KUKA KRL program: Rack_Verde_Dejar.src, Rack_Verde_Dejar.dat

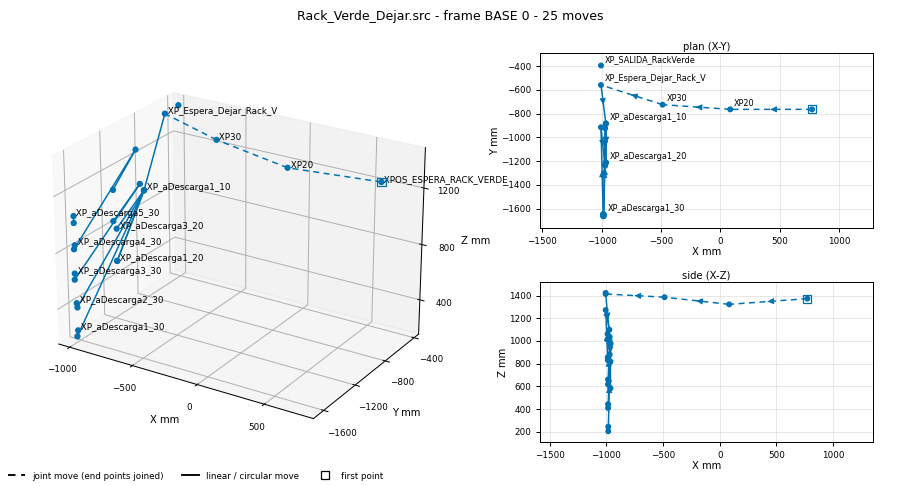
[picture p0: tool path of Rack_Verde_Dejar.src in frame BASE 0, 25 of 38 moves have a stored position in this frame; points joined in program order, loops and branches not executed]
--- Rack_Verde_Dejar.src ---
&ACCESS RVO1
&REL 3309
&COMMENT DEJAR BAT EN RACK VERDE
&PARAM EDITMASK = *
&PARAM TEMPLATE = C:\KRC\Roboter\Template\vorgabe
&PARAM DISKPATH = KRC:\R1\Program\MAFELEC
DEF Rack_Verde_Dejar( )
;FOLD INI;%{PE}
;FOLD BASISTECH INI
    GLOBAL INTERRUPT DECL 3 WHEN $STOPMESS==TRUE DO IR_STOPM ( )
    INTERRUPT ON 3
    BAS (#INITMOV,0 )
  ;ENDFOLD (BASISTECH INI)
;FOLD SPOTTECH INI
USERSPOT(#INIT)
;ENDFOLD (SPOTTECH INI)
;FOLD GRIPPERTECH INI
USER_GRP(0,DUMMY,DUMMY,GDEFAULT)
;ENDFOLD (GRIPPERTECH INI)
;FOLD USER INI
GIRO_A_P=FALSE
GIRO_A_N=FALSE
GIRO_B_P=FALSE
GIRO_B_N=FALSE
GIRO_C_P=FALSE
GIRO_C_N=FALSE
INTERRUPT DECL 26 WHEN I_121R1S102 OR I_121R1S202 DO PARO_RAPIDO ()
INTERRUPT DECL 27 WHEN I_121R1S302 OR I_121R1S402 DO PARO_RAPIDO ()
O_TYPE_INFO=0
SELECT_T1=FALSE

  ;ENDFOLD (USER INI)
;ENDFOLD (INI)
;################################################
; PROYECTO: MAFELEC PLANTA DE BATERIAS
; ROBOT: 121_R1
; PROGRAMA: DESCARGA DE BATERIA EN RACK VERDE
; CREADO POR: Tu amigo y vecino Spiderman(zaisor robotics)
; FECHA: 23-NOVIEMBRE-2022
; MODIFICADO POR:
; FECHA MODIFICACION: 17-ENERO-2023
;################################################

; FOLD CARGA VALORES DE POSICION

XP_DEJAR_VERDE=FRAME_POS
XP_DEJAR_VERDE.z=FRAME_POS.z+3
XP_DROP_1=XP_DEJAR_VERDE
XP_DROP_2=XP_DEJAR_VERDE
XP_DROP_3=XP_DEJAR_VERDE
XP_DROP_4=XP_DEJAR_VERDE
XP_DROP_5=XP_DEJAR_VERDE

XP_DROP_1.z=XP_DROP_1.z + 80
XP_DROP_2.z=XP_DROP_2.z + 80
XP_DROP_3.z=XP_DROP_3.z + 80
XP_DROP_4.z=XP_DROP_4.z + 80
XP_DROP_5.z=XP_DROP_5.z + 80
;ENDFOLD

;FOLD PTP POS_ESPERA_RACK_VERDE Vel=100 % H Tool[11]:T_Gripper1_Carga Base[0];%{PE}%R 8.3.48,%MKUKATPBASIS,%CMOVE,%VPTP,%P 1:PTP, 2:POS_ESPERA_RACK_VERDE, 3:, 5:100, 7:H
$BWDSTART=FALSE
PDAT_ACT=PH
FDAT_ACT=FPOS_ESPERA_RACK_VERDE
BAS(#PTP_PARAMS,100)
PTP XPOS_ESPERA_RACK_VERDE
;ENDFOLD
;ESPERA AREA 1
WAIT FOR I_ARDY_1
O_AREL_1=FALSE

Empujador(1,"R",TRUE)
Empujador(2,"R",TRUE)

;FOLD PTP P20 CONT Vel=100 % M Tool[11]:T_Gripper1_Carga Base[0];%{PE}%R 8.3.48,%MKUKATPBASIS,%CMOVE,%VPTP,%P 1:PTP, 2:P20, 3:C_DIS, 5:100, 7:M
$BWDSTART=FALSE
PDAT_ACT=PM
FDAT_ACT=FP20
BAS(#PTP_PARAMS,100)
PTP XP20 C_DIS
;ENDFOLD
;FOLD PTP P30 CONT Vel=100 % M Tool[11]:T_Gripper1_Carga Base[0];%{PE}%R 8.3.48,%MKUKATPBASIS,%CMOVE,%VPTP,%P 1:PTP, 2:P30, 3:C_DIS, 5:100, 7:M
$BWDSTART=FALSE
PDAT_ACT=PM
FDAT_ACT=FP30
BAS(#PTP_PARAMS,100)
PTP XP30 C_DIS
;ENDFOLD

; POSICION DE ESPERA A DEJAR BATERIA EN RACK VERDE
;FOLD PTP P_Espera_Dejar_Rack_V Vel=100 % L Tool[11]:T_Gripper1_Carga Base[0];%{PE}%R 8.3.48,%MKUKATPBASIS,%CMOVE,%VPTP,%P 1:PTP, 2:P_Espera_Dejar_Rack_V, 3:, 5:100, 7:L
$BWDSTART=FALSE
PDAT_ACT=PL
FDAT_ACT=FP_Espera_Dejar_Rack_V
BAS(#PTP_PARAMS,100)
PTP XP_Espera_Dejar_Rack_V
;ENDFOLD

; FOLD ACTIVA VIGILANCIA SOBREPASO
;INTERRUPT ON 26
;INTERRUPT ON 27
;ENDFOLD

;CONTROL DE AUSENCIA DE PIEZA EN GRIPPER
IF (I_SIMULACION==FALSE) THEN
IF NOT I_121R1S1000 THEN
HALT
ENDIF
ENDIF

;CONTROL APERTURA GRIPPER

IF (I_121R1S131A==FALSE) OR (I_121R1S132A==FALSE) OR (I_121R1S133A==FALSE) OR (I_121R1S134A==FALSE) THEN
HALT
ENDIF

IF PGNO==11 THEN
O_TYPE_RQ=TRUE
WAIT FOR (I_TYPE_INFO>10) AND (I_TYPE_INFO<16)
RV_Bandeja_Nr=I_TYPE_INFO
O_TYPE_RQ=FALSE
ENDIF

WAIT FOR (RV_Bandeja_Nr>10) AND (RV_Bandeja_Nr<16)

SWITCH RV_Bandeja_Nr ;

CASE 11
; MOVIMIENTOS HACIA BANDEJA 1
O_TYPE_INFO=11

WAIT FOR I_Rack1_S1==TRUE
;FOLD LIN P_aDescarga1_10 CONT Vel=0.5 m/s L Tool[11]:T_Gripper1_Carga Base[0];%{PE}%R 8.3.48,%MKUKATPBASIS,%CMOVE,%VLIN,%P 1:LIN, 2:P_aDescarga1_10, 3:C_DIS C_DIS, 5:0.5, 7:L
$BWDSTART=FALSE
LDAT_ACT=LL
FDAT_ACT=FP_aDescarga1_10
BAS(#CP_PARAMS,0.5)
LIN XP_aDescarga1_10 C_DIS C_DIS
;ENDFOLD
;FOLD LIN P_aDescarga1_20 CONT Vel=0.5 m/s L Tool[11]:T_Gripper1_Carga Base[0];%{PE}%R 8.3.48,%MKUKATPBASIS,%CMOVE,%VLIN,%P 1:LIN, 2:P_aDescarga1_20, 3:C_DIS C_DIS, 5:0.5, 7:L
$BWDSTART=FALSE
LDAT_ACT=LL
FDAT_ACT=FP_aDescarga1_20
BAS(#CP_PARAMS,0.5)
LIN XP_aDescarga1_20 C_DIS C_DIS
;ENDFOLD
O_LIMITS_OK=TRUE
O_LIMITS_NOK=FALSE

IF (O_INPICKER_OK==TRUE) AND (O_INPICKER_NOK==FALSE) AND (O_LIMITS_OK==TRUE) AND (O_LIMITS_NOK==FALSE) THEN
; #### MOVIMIENTOS A DESCARGA CONTROLADOS POR ####
; #### LA CAMARA DE VISION                    ####

;FOLD LIN P_DROP_1 Vel=0.3 m/s L Tool[11]:T_Gripper1_Carga Base[0];%{PE}%R 8.3.48,%MKUKATPBASIS,%CMOVE,%VLIN,%P 1:LIN, 2:P_DROP_1, 3:, 5:0.3, 7:L
$BWDSTART=FALSE
LDAT_ACT=LL
FDAT_ACT=FP_DROP_1
BAS(#CP_PARAMS,0.3)
LIN XP_DROP_1
;ENDFOLD
;FOLD LIN P_DEJAR_VERDE Vel=0.1 m/s L Tool[11]:T_Gripper1_Carga Base[0];%{PE}%R 8.3.48,%MKUKATPBASIS,%CMOVE,%VLIN,%P 1:LIN, 2:P_DEJAR_VERDE, 3:, 5:0.1, 7:L
$BWDSTART=FALSE
LDAT_ACT=LL
FDAT_ACT=FP_DEJAR_VERDE
BAS(#CP_PARAMS,0.1)
LIN XP_DEJAR_VERDE
;ENDFOLD

ELSE

; #### MOVIMIENTOS A DESCARGA CONTROLADOS POR ####
; #### EL OPERARIO                            ####
;FOLD ESPERA LLAVE SELECTORA EN MODO T1
WAIT FOR $T1
SELECT_T1=TRUE
;ENDFOLD
;FOLD LIN P_aDescarga1_30 CONT Vel=0.2 m/s L Tool[11]:T_Gripper1_Carga Base[0];%{PE}%R 8.3.48,%MKUKATPBASIS,%CMOVE,%VLIN,%P 1:LIN, 2:P_aDescarga1_30, 3:C_DIS C_DIS, 5:0.2, 7:L
$BWDSTART=FALSE
LDAT_ACT=LL
FDAT_ACT=FP_aDescarga1_30
BAS(#CP_PARAMS,0.2)
LIN XP_aDescarga1_30 C_DIS C_DIS
;ENDFOLD

;POSICION DE DESCARGA 1
;CUIDADO CON EL LINEAL NO EJECUTARLO HASTA EL FINAL
;POSIBILIDAD DE COLISION
;EN ESTE PUNTO LLEVAR EL ROBOT HASTA LA DESCARGA DE BANDEJA
;UNA VEZ TENEMOS EL ROBOT YA EN LA POSICION DE DEJADA TENEMOS
;QUE ACTIVAR LAS SALIDAS DE LAS CLAMPAS PARA DEJAR LA BATERIA
;SALIDA 246 O_121R1Y13A PINES BLOQUEO ADELANTE ESTARA EN 1 PONERLA A 0
;SEGUIDAMENTE LA SALIDA 245 O_121R1Y13B PINES BLOQUEO ATRAS ESTARA A 0 PONERLA A 1
;AL ABRIR LOS PINES DE LAS CLAMPAS EL SIGUIENTE PASO ES SELECCIONAR LA LINEA
;ENDIF Y CONTINUAR PROGRAMA
;FOLD LIN Rack_Verde_Pos1 Vel=0.2 m/s L Tool[11]:T_Gripper1_Carga Base[0];%{PE}%R 8.3.48,%MKUKATPBASIS,%CMOVE,%VLIN,%P 1:LIN, 2:Rack_Verde_Pos1, 3:, 5:0.2, 7:L
$BWDSTART=FALSE
LDAT_ACT=LL
FDAT_ACT=FRack_Verde_Pos1
BAS(#CP_PARAMS,0.2)
LIN XRack_Verde_Pos1
;ENDFOLD
ENDIF

CASE 12
; MOVIMIENTOS HACIA BANDEJA 2
O_TYPE_INFO=12
WAIT FOR I_Rack1_S2==TRUE
;FOLD LIN P_aDescarga2_10 CONT Vel=0.5 m/s L Tool[11]:T_Gripper1_Carga Base[0];%{PE}%R 8.3.48,%MKUKATPBASIS,%CMOVE,%VLIN,%P 1:LIN, 2:P_aDescarga2_10, 3:C_DIS C_DIS, 5:0.5, 7:L
$BWDSTART=FALSE
LDAT_ACT=LL
FDAT_ACT=FP_aDescarga2_10
BAS(#CP_PARAMS,0.5)
LIN XP_aDescarga2_10 C_DIS C_DIS
;ENDFOLD
;FOLD LIN P_aDescarga2_20 CONT Vel=0.5 m/s L Tool[11]:T_Gripper1_Carga Base[0];%{PE}%R 8.3.48,%MKUKATPBASIS,%CMOVE,%VLIN,%P 1:LIN, 2:P_aDescarga2_20, 3:C_DIS C_DIS, 5:0.5, 7:L
$BWDSTART=FALSE
LDAT_ACT=LL
FDAT_ACT=FP_aDescarga2_20
BAS(#CP_PARAMS,0.5)
LIN XP_aDescarga2_20 C_DIS C_DIS
;ENDFOLD

IF (O_INPICKER_OK==TRUE) AND (O_INPICKER_NOK==FALSE) AND (O_LIMITS_OK==TRUE) AND (O_LIMITS_NOK==FALSE) THEN
; #### MOVIMIENTOS A DESCARGA CONTROLADOS POR ####
; #### LA CAMARA DE VISION                    ####

;FOLD LIN P_DROP_2 Vel=0.3 m/s L Tool[11]:T_Gripper1_Carga Base[0];%{PE}%R 8.3.48,%MKUKATPBASIS,%CMOVE,%VLIN,%P 1:LIN, 2:P_DROP_2, 3:, 5:0.3, 7:L
$BWDSTART=FALSE
LDAT_ACT=LL
FDAT_ACT=FP_DROP_2
BAS(#CP_PARAMS,0.3)
LIN XP_DROP_2
;ENDFOLD
;FOLD LIN P_DEJAR_VERDE Vel=0.1 m/s L Tool[11]:T_Gripper1_Carga Base[0];%{PE}%R 8.3.48,%MKUKATPBASIS,%CMOVE,%VLIN,%P 1:LIN, 2:P_DEJAR_VERDE, 3:, 5:0.1, 7:L
$BWDSTART=FALSE
LDAT_ACT=LL
FDAT_ACT=FP_DEJAR_VERDE
BAS(#CP_PARAMS,0.1)
LIN XP_DEJAR_VERDE
;ENDFOLD

ELSE
; #### MOVIMIENTOS A DESCARGA CONTROLADOS POR ####
; #### EL OPERARIO                            ####
;FOLD ESPERA LLAVE SELECTORA EN MODO T1
WAIT FOR $T1
SELECT_T1=TRUE
;ENDFOLD
;FOLD LIN P_aDescarga2_30 CONT Vel=0.2 m/s L Tool[11]:T_Gripper1_Carga Base[0];%{PE}%R 8.3.48,%MKUKATPBASIS,%CMOVE,%VLIN,%P 1:LIN, 2:P_aDescarga2_30, 3:C_DIS C_DIS, 5:0.2, 7:L
$BWDSTART=FALSE
LDAT_ACT=LL
FDAT_ACT=FP_aDescarga2_30
BAS(#CP_PARAMS,0.2)
LIN XP_aDescarga2_30 C_DIS C_DIS
;ENDFOLD

;POSICION DE DESCARGA 2
;CUIDADO CON EL LINEAL NO EJECUTARLO HASTA EL FINAL
;POSIBILIDAD DE COLISION
;EN ESTE PUNTO LLEVAR EL ROBOT HASTA LA DESCARGA DE BANDEJA
;UNA VEZ TENEMOS EL ROBOT YA EN LA POSICION DE DEJADA TENEMOS
;QUE ACTIVAR LAS SALIDAS DE LAS CLAMPAS PARA DEJAR LA BATERIA
;SALIDA 246 O_121R1Y13A PINES BLOQUEO ADELANTE ESTARA EN 1 PONERLA A 0
;SEGUIDAMENTE LA SALIDA 245 O_121R1Y13B PINES BLOQUEO ATRAS ESTARA A 0 PONERLA A 1
;AL ABRIR LOS PINES DE LAS CLAMPAS EL SIGUIENTE PASO ES SELECCIONAR LA LINEA
;ENDIF Y CONTINUAR PROGRAMA
;FOLD LIN Rack_Verde_Pos2 Vel=0.2 m/s L Tool[11]:T_Gripper1_Carga Base[0];%{PE}%R 8.3.48,%MKUKATPBASIS,%CMOVE,%VLIN,%P 1:LIN, 2:Rack_Verde_Pos2, 3:, 5:0.2, 7:L
$BWDSTART=FALSE
LDAT_ACT=LL
FDAT_ACT=FRack_Verde_Pos2
BAS(#CP_PARAMS,0.2)
LIN XRack_Verde_Pos2
;ENDFOLD
ENDIF

CASE 13
; MOVIMIENTOS HACIA BANDEJA 3
O_TYPE_INFO=13
WAIT FOR I_Rack1_S3==TRUE
;FOLD LIN P_aDescarga3_10 CONT Vel=0.5 m/s L Tool[11]:T_Gripper1_Carga Base[0];%{PE}%R 8.3.48,%MKUKATPBASIS,%CMOVE,%VLIN,%P 1:LIN, 2:P_aDescarga3_10, 3:C_DIS C_DIS, 5:0.5, 7:L
$BWDSTART=FALSE
LDAT_ACT=LL
FDAT_ACT=FP_aDescarga3_10
BAS(#CP_PARAMS,0.5)
LIN XP_aDescarga3_10 C_DIS C_DIS
;ENDFOLD
;FOLD LIN P_aDescarga3_20 CONT Vel=0.5 m/s L Tool[11]:T_Gripper1_Carga Base[0];%{PE}%R 8.3.48,%MKUKATPBASIS,%CMOVE,%VLIN,%P 1:LIN, 2:P_aDescarga3_20, 3:C_DIS C_DIS, 5:0.5, 7:L
$BWDSTART=FALSE
LDAT_ACT=LL
FDAT_ACT=FP_aDescarga3_20
BAS(#CP_PARAMS,0.5)
LIN XP_aDescarga3_20 C_DIS C_DIS
;ENDFOLD


IF (O_INPICKER_OK==TRUE) AND (O_INPICKER_NOK==FALSE) AND (O_LIMITS_OK==TRUE) AND (O_LIMITS_NOK==FALSE) THEN
; #### MOVIMIENTOS A DESCARGA CONTROLADOS POR ####
; #### LA CAMARA DE VISION                    ####

;FOLD LIN P_DROP_3 Vel=0.3 m/s L Tool[11]:T_Gripper1_Carga Base[0];%{PE}%R 8.3.48,%MKUKATPBASIS,%CMOVE,%VLIN,%P 1:LIN, 2:P_DROP_3, 3:, 5:0.3, 7:L
$BWDSTART=FALSE
LDAT_ACT=LL
FDAT_ACT=FP_DROP_3
BAS(#CP_PARAMS,0.3)
LIN XP_DROP_3
;ENDFOLD
;FOLD LIN P_DEJAR_VERDE Vel=0.1 m/s L Tool[11]:T_Gripper1_Carga Base[0];%{PE}%R 8.3.48,%MKUKATPBASIS,%CMOVE,%VLIN,%P 1:LIN, 2:P_DEJAR_VERDE, 3:, 5:0.1, 7:L
$BWDSTART=FALSE
LDAT_ACT=LL
FDAT_ACT=FP_DEJAR_VERDE
BAS(#CP_PARAMS,0.1)
LIN XP_DEJAR_VERDE
;ENDFOLD

ELSE
; #### MOVIMIENTOS A DESCARGA CONTROLADOS POR ####
; #### EL OPERARIO                            ####
;FOLD ESPERA LLAVE SELECTORA EN MODO T1
WAIT FOR $T1
SELECT_T1=TRUE
;ENDFOLD
;FOLD LIN P_aDescarga3_30 CONT Vel=0.2 m/s L Tool[11]:T_Gripper1_Carga Base[0];%{PE}%R 8.3.48,%MKUKATPBASIS,%CMOVE,%VLIN,%P 1:LIN, 2:P_aDescarga3_30, 3:C_DIS C_DIS, 5:0.2, 7:L
$BWDSTART=FALSE
LDAT_ACT=LL
FDAT_ACT=FP_aDescarga3_30
BAS(#CP_PARAMS,0.2)
LIN XP_aDescarga3_30 C_DIS C_DIS
;ENDFOLD

;POSICION DE DESCARGA 3
;CUIDADO CON EL LINEAL NO EJECUTARLO HASTA EL FINAL
;POSIBILIDAD DE COLISION
;EN ESTE PUNTO LLEVAR EL ROBOT HASTA LA DESCARGA DE BANDEJA
;UNA VEZ TENEMOS EL ROBOT YA EN LA POSICION DE DEJADA TENEMOS
;QUE ACTIVAR LAS SALIDAS DE LAS CLAMPAS PARA DEJAR LA BATER
;SALIDA 246 y 248 PINES BLOQUEO ADELANTE ESTARA EN 1 PONERLA A 0
;SEGUIDAMENTE LA SALIDA 245 y 247 PINES BLOQUEO ATRAS ESTARA A 0 PONERLA A 1
;AL ABRIR LOS PINES DE LAS CLAMPAS EL SIGUIENTE PASO ES SELECCIONAR LA LINEA
;ENDIF Y CONTINUAR PROGRAMA
;FOLD LIN Rack_Verde_Pos3 Vel=0.2 m/s L Tool[11]:T_Gripper1_Carga Base[0];%{PE}%R 8.3.48,%MKUKATPBASIS,%CMOVE,%VLIN,%P 1:LIN, 2:Rack_Verde_Pos3, 3:, 5:0.2, 7:L
$BWDSTART=FALSE
LDAT_ACT=LL
FDAT_ACT=FRack_Verde_Pos3
BAS(#CP_PARAMS,0.2)
LIN XRack_Verde_Pos3
;ENDFOLD
ENDIF

CASE 14
; MOVIMIENTOS HACIA BANDEJA4
O_TYPE_INFO=14
WAIT FOR I_Rack1_S4==TRUE
;FOLD LIN P_aDescarga4_10 CONT Vel=0.5 m/s L Tool[11]:T_Gripper1_Carga Base[0];%{PE}%R 8.3.48,%MKUKATPBASIS,%CMOVE,%VLIN,%P 1:LIN, 2:P_aDescarga4_10, 3:C_DIS C_DIS, 5:0.5, 7:L
$BWDSTART=FALSE
LDAT_ACT=LL
FDAT_ACT=FP_aDescarga4_10
BAS(#CP_PARAMS,0.5)
LIN XP_aDescarga4_10 C_DIS C_DIS
;ENDFOLD
;FOLD LIN P_aDescarga4_20 CONT Vel=0.5 m/s L Tool[11]:T_Gripper1_Carga Base[0];%{PE}%R 8.3.48,%MKUKATPBASIS,%CMOVE,%VLIN,%P 1:LIN, 2:P_aDescarga4_20, 3:C_DIS C_DIS, 5:0.5, 7:L
$BWDSTART=FALSE
LDAT_ACT=LL
FDAT_ACT=FP_aDescarga4_20
BAS(#CP_PARAMS,0.5)
LIN XP_aDescarga4_20 C_DIS C_DIS
;ENDFOLD

IF (O_INPICKER_OK==TRUE) AND (O_INPICKER_NOK==FALSE) AND (O_LIMITS_OK==TRUE) AND (O_LIMITS_NOK==FALSE) THEN
; #### MOVIMIENTOS A DESCARGA CONTROLADOS POR ####
; #### LA CAMARA DE VISION                    ####

;FOLD LIN P_DROP_4 Vel=0.3 m/s L Tool[11]:T_Gripper1_Carga Base[0];%{PE}%R 8.3.48,%MKUKATPBASIS,%CMOVE,%VLIN,%P 1:LIN, 2:P_DROP_4, 3:, 5:0.3, 7:L
$BWDSTART=FALSE
LDAT_ACT=LL
FDAT_ACT=FP_DROP_4
BAS(#CP_PARAMS,0.3)
LIN XP_DROP_4
;ENDFOLD
;FOLD LIN P_DEJAR_VERDE Vel=0.1 m/s L Tool[11]:T_Gripper1_Carga Base[0];%{PE}%R 8.3.48,%MKUKATPBASIS,%CMOVE,%VLIN,%P 1:LIN, 2:P_DEJAR_VERDE, 3:, 5:0.1, 7:L
$BWDSTART=FALSE
LDAT_ACT=LL
FDAT_ACT=FP_DEJAR_VERDE
BAS(#CP_PARAMS,0.1)
LIN XP_DEJAR_VERDE
;ENDFOLD

ELSE
; #### MOVIMIENTOS A DESCARGA CONTROLADOS POR ####
; #### EL OPERARIO                            ####
;FOLD ESPERA LLAVE SELECTORA EN MODO T1
WAIT FOR $T1
SELECT_T1=TRUE
;ENDFOLD
;FOLD LIN P_aDescarga4_30 CONT Vel=0.2 m/s L Tool[11]:T_Gripper1_Carga Base[0];%{PE}%R 8.3.48,%MKUKATPBASIS,%CMOVE,%VLIN,%P 1:LIN, 2:P_aDescarga4_30, 3:C_DIS C_DIS, 5:0.2, 7:L
$BWDSTART=FALSE
LDAT_ACT=LL
FDAT_ACT=FP_aDescarga4_30
BAS(#CP_PARAMS,0.2)
LIN XP_aDescarga4_30 C_DIS C_DIS
;ENDFOLD

;POSICION DE DESCARGA 4
;CUIDADO CON EL LINEAL NO EJECUTARLO HASTA EL FINAL
;POSIBILIDAD DE COLISION
;EN ESTE PUNTO LLEVAR EL ROBOT HASTA LA DESCARGA DE BANDEJA
;UNA VEZ TENEMOS EL ROBOT YA EN LA POSICION DE DEJADA TENEMOS
;QUE ACTIVAR LAS SALIDAS DE LAS CLAMPAS PARA DEJAR LA BATERIA
;SALIDA 246 y 248 PINES BLOQUEO ADELANTE ESTARA EN 1 PONERLA A 0
;SEGUIDAMENTE LA SALIDA 245 y 247 PINES BLOQUEO ATRAS ESTARA A 0 PONERLA A 1
;AL ABRIR LOS PINES DE LAS CLAMPAS EL SIGUIENTE PASO ES SELECCIONAR LA LINEA
;ENDIF Y CONTINUAR PROGRAMA
;FOLD LIN Rack_Verde_Pos4 Vel=0.2 m/s L Tool[11]:T_Gripper1_Carga Base[0];%{PE}%R 8.3.48,%MKUKATPBASIS,%CMOVE,%VLIN,%P 1:LIN, 2:Rack_Verde_Pos4, 3:, 5:0.2, 7:L
$BWDSTART=FALSE
LDAT_ACT=LL
FDAT_ACT=FRack_Verde_Pos4
BAS(#CP_PARAMS,0.2)
LIN XRack_Verde_Pos4
;ENDFOLD
ENDIF

CASE 15
; MOVIMIENTOS HACIA BANDEJA 5
O_TYPE_INFO=15
WAIT FOR I_Rack1_S5==TRUE
;FOLD LIN P_aDescarga5_10 CONT Vel=0.5 m/s L Tool[11]:T_Gripper1_Carga Base[0];%{PE}%R 8.3.48,%MKUKATPBASIS,%CMOVE,%VLIN,%P 1:LIN, 2:P_aDescarga5_10, 3:C_DIS C_DIS, 5:0.5, 7:L
$BWDSTART=FALSE
LDAT_ACT=LL
FDAT_ACT=FP_aDescarga5_10
BAS(#CP_PARAMS,0.5)
LIN XP_aDescarga5_10 C_DIS C_DIS
;ENDFOLD
;FOLD LIN P_aDescarga5_20 CONT Vel=0.5 m/s L Tool[11]:T_Gripper1_Carga Base[0];%{PE}%R 8.3.48,%MKUKATPBASIS,%CMOVE,%VLIN,%P 1:LIN, 2:P_aDescarga5_20, 3:C_DIS C_DIS, 5:0.5, 7:L
$BWDSTART=FALSE
LDAT_ACT=LL
FDAT_ACT=FP_aDescarga5_20
BAS(#CP_PARAMS,0.5)
LIN XP_aDescarga5_20 C_DIS C_DIS
;ENDFOLD

IF (O_INPICKER_OK==TRUE) AND (O_INPICKER_NOK==FALSE) AND (O_LIMITS_OK==TRUE) AND (O_LIMITS_NOK==FALSE) THEN
; #### MOVIMIENTOS A DESCARGA CONTROLADOS POR ####
; #### LA CAMARA DE VISION                    ####

;FOLD LIN P_DROP_5 Vel=0.3 m/s L Tool[11]:T_Gripper1_Carga Base[0];%{PE}%R 8.3.48,%MKUKATPBASIS,%CMOVE,%VLIN,%P 1:LIN, 2:P_DROP_5, 3:, 5:0.3, 7:L
$BWDSTART=FALSE
LDAT_ACT=LL
FDAT_ACT=FP_DROP_5
BAS(#CP_PARAMS,0.3)
LIN XP_DROP_5
;ENDFOLD
;FOLD LIN P_DEJAR_VERDE Vel=0.1 m/s L Tool[11]:T_Gripper1_Carga Base[0];%{PE}%R 8.3.48,%MKUKATPBASIS,%CMOVE,%VLIN,%P 1:LIN, 2:P_DEJAR_VERDE, 3:, 5:0.1, 7:L
$BWDSTART=FALSE
LDAT_ACT=LL
FDAT_ACT=FP_DEJAR_VERDE
BAS(#CP_PARAMS,0.1)
LIN XP_DEJAR_VERDE
;ENDFOLD

ELSE
; #### MOVIMIENTOS A DESCARGA CONTROLADOS POR ####
; #### EL OPERARIO                            ####
;FOLD ESPERA LLAVE SELECTORA EN MODO T1
WAIT FOR $T1
SELECT_T1=TRUE
;ENDFOLD
;FOLD LIN P_aDescarga5_30 CONT Vel=0.2 m/s L Tool[11]:T_Gripper1_Carga Base[0];%{PE}%R 8.3.48,%MKUKATPBASIS,%CMOVE,%VLIN,%P 1:LIN, 2:P_aDescarga5_30, 3:C_DIS C_DIS, 5:0.2, 7:L
$BWDSTART=FALSE
LDAT_ACT=LL
FDAT_ACT=FP_aDescarga5_30
BAS(#CP_PARAMS,0.2)
LIN XP_aDescarga5_30 C_DIS C_DIS
;ENDFOLD

;POSICION DE DESCARGA 5
;CUIDADO CON EL LINEAL NO EJECUTARLO HASTA EL FINAL
;POSIBILIDAD DE COLISION
;EN ESTE PUNTO LLEVAR EL ROBOT HASTA LA DESCARGA DE BANDEJA
;UNA VEZ TENEMOS EL ROBOT YA EN LA POSICION DE DEJADA TENEMOS
;QUE ACTIVAR LAS SALIDAS DE LAS CLAMPAS PARA DEJAR LA BATERIA
;SALIDA 246 O_121R1Y13A PINES BLOQUEO ADELANTE ESTARA EN 1 PONERLA A 0
;SEGUIDAMENTE LA SALIDA 245 O_121R1Y13B PINES BLOQUEO ATRAS ESTARA A 0 PONERLA A 1
;AL ABRIR LOS PINES DE LAS CLAMPAS EL SIGUIENTE PASO ES SELECCIONAR LA LINEA
;ENDIF Y CONTINUAR PROGRAMA
;FOLD LIN Rack_Verde_Pos5 Vel=0.2 m/s L Tool[11]:T_Gripper1_Carga Base[0];%{PE}%R 8.3.48,%MKUKATPBASIS,%CMOVE,%VLIN,%P 1:LIN, 2:Rack_Verde_Pos5, 3:, 5:0.2, 7:L
$BWDSTART=FALSE
LDAT_ACT=LL
FDAT_ACT=FRack_Verde_Pos5
BAS(#CP_PARAMS,0.2)
LIN XRack_Verde_Pos5
;ENDFOLD
ENDIF

DEFAULT
HALT
HALT
; #### CODIGO DE DESCARGA ERRONEO ####
HALT
BRAKE
ENDSWITCH

; FOLD MOVIMIENTOS DE SALIDA RACK VERDE
INI_DROP:
GIRO_A_P=FALSE
GIRO_A_N=FALSE
GIRO_B_P=FALSE
GIRO_B_N=FALSE
GIRO_C_P=FALSE
GIRO_C_N=FALSE

PTP $POS_ACT

IF (I_SIMULACION==FALSE) THEN

Repite=0

WHILE (I_121R1S102==TRUE) OR (I_121R1S202==TRUE) OR (I_121R1S302==TRUE) OR (I_121R1S402==TRUE)

Repite=Repite+1
LIN_REL{Z +1}
WAIT SEC 0.1

IF Repite>=3 THEN
HALT
; SUPERADO NUMERO DE REPETICIONES
HALT
ENDIF

ENDWHILE

Repite=0

WHILE (I_121R1S101==FALSE) AND (I_121R1S201==FALSE) AND (I_121R1S301==FALSE) AND (I_121R1S401==FALSE)
IF (I_121R1S102==TRUE) OR (I_121R1S202==TRUE) OR (I_121R1S302==TRUE) OR (I_121R1S402==TRUE) THEN
HALT
HALT
HALT
ENDIF
Repite=Repite+1
LIN_REL{Z -1}
WAIT SEC 0.1

IF Repite>=8 THEN
HALT
; SUPERADO NUMERO DE REPETICIONES
HALT
ENDIF

;PARA ABRIR PINES DE LA BATERIA SALIDA O_121R1Y13B
;GOTO ctrl_dejar
ENDWHILE

; #### CONTROL DE PRESENCIA PARA ABRIR ####
WAIT FOR (I_121R1S101==TRUE) OR (I_121R1S301==TRUE) OR (I_121R1S201==TRUE) OR (I_121R1S401==TRUE)
fin_dejar:
ENDIF

O_INPICKER_OK=FALSE
O_INPICKER_NOK=FALSE
O_LIMITS_OK=FALSE
O_LIMITS_NOK=FALSE
O_LIMIT_X=FALSE
O_LIMIT_Y=FALSE
O_LIMIT_Z=FALSE
O_LIMIT_A=FALSE
O_LIMIT_B=FALSE
O_LIMIT_C=FALSE

PTP $POS_ACT
PINES("R")

PTP $POS_ACT
WAIT FOR $EXT; CAMBIAR LA LLAVE A MODO EXT

LIN_REL{Z +100}
O_JRDY_2=TRUE
BAS(#CP_PARAMS,1.5)

; #### CONTROL DE AUSENCIA DE BATERIA ####
WAIT FOR NOT I_121R1S1000

LIN_REL{Y 300,Z +100} C_DIS
LIN_REL{Y 400,Z +350} C_DIS
; ENDFOLD
; FOLD FIN VIGILANCIA SOBREPASO
INTERRUPT OFF 26
INTERRUPT OFF 27
;ENDFOLD

;FOLD LIN P_SALIDA_RackVerde Vel=1 m/s M Tool[9]:T_Gripper1_Vacio Base[0];%{PE}%R 8.3.48,%MKUKATPBASIS,%CMOVE,%VLIN,%P 1:LIN, 2:P_SALIDA_RackVerde, 3:, 5:1, 7:M
$BWDSTART=FALSE
LDAT_ACT=LM
FDAT_ACT=FP_SALIDA_RackVerde
BAS(#CP_PARAMS,1)
LIN XP_SALIDA_RackVerde
;ENDFOLD




Rack_Verde_Cerrar_D()

;TRABAJO REALIZADO
O_JRDY_4 = TRUE

END
DEF Descarga_B1()
END
DEF Descarga_B2()
END
DEF Descarga_B3()
END
DEF Descarga_B4()
END
DEF Descarga_B5()
END
DEF PARO_RAPIDO ()
BRAKE F
END

--- Rack_Verde_Dejar.dat ---
&ACCESS RVO1
&REL 3309
&COMMENT DEJAR BAT EN RACK VERDE
&PARAM EDITMASK = *
&PARAM TEMPLATE = C:\KRC\Roboter\Template\vorgabe
&PARAM DISKPATH = KRC:\R1\Program\MAFELEC
DEFDAT  Rack_Verde_Dejar
;FOLD EXTERNAL DECLARATIONS;%{PE}%MKUKATPBASIS,%CEXT,%VCOMMON,%P
;FOLD GRIPPERTECH EXT
EXT  H50 (INT  :IN,INT  :IN,INT  :IN,GRP_TYP  :IN )
;ENDFOLD (GRIPPERTECH EXT)
;FOLD SPOTTECH EXT
EXT  USERSPOT (S_COMMAND  :IN,SPOT_TYPE  :IN )
;ENDFOLD (SPOTTECH EXT)
;FOLD BASISTECH EXT;%{PE}%MKUKATPBASIS,%CEXT,%VEXT,%P
EXT  BAS (BAS_COMMAND  :IN,REAL  :IN )
DECL INT SUCCESS
;ENDFOLD (BASISTECH EXT)
;FOLD USER EXT;%{E}%MKUKATPUSER,%CEXT,%VEXT,%P
;Make your modifications here

;ENDFOLD (USER EXT)
;ENDFOLD (EXTERNAL DECLARATIONS)
DECL BASIS_SUGG_T LAST_BASIS={POINT1[] "P_DEJAR_AUTO            ",POINT2[] "P_DEJAR_AUTO            ",CP_PARAMS[] "L                       ",PTP_PARAMS[] "H                       ",CONT[] "                        ",CP_VEL[] "0.1                     ",PTP_VEL[] "100                     ",SYNC_PARAMS[] "SYNCDAT                 ",SPL_NAME[] "S0                      ",A_PARAMS[] "ADAT0                   "}
DECL PDAT PH={VEL 100.000,ACC 100.000,APO_DIST 100.000,APO_MODE #CDIS,GEAR_JERK 50.0000,EXAX_IGN 0}
DECL E6POS XPOS_ESPERA_DROP_RACK1={X -1005.21851,Y -395.575073,Z 1423.46069,A -87.1007538,B -0.167297319,C 179.537186,S 2,T 42,E1 0.0,E2 0.0,E3 0.0,E4 0.0,E5 0.0,E6 0.0}
DECL FDAT FPOS_ESPERA_DROP_RACK1={TOOL_NO 11,BASE_NO 0,IPO_FRAME #BASE,POINT2[] " ",TQ_STATE FALSE}
DECL E6POS XP10={X 772.101379,Y -764.727417,Z 1373.18774,A -87.1007538,B -0.167297110,C 179.537186,S 2,T 34,E1 0.0,E2 0.0,E3 0.0,E4 0.0,E5 0.0,E6 0.0}
DECL FDAT FP10={TOOL_NO 11,BASE_NO 0,IPO_FRAME #BASE,POINT2[] " ",TQ_STATE FALSE}
DECL E6POS XP20={X 83.1755524,Y -764.726563,Z 1322.80212,A -87.1007538,B -0.167296991,C 179.537186,S 2,T 34,E1 0.0,E2 0.0,E3 0.0,E4 0.0,E5 0.0,E6 0.0}
DECL FDAT FP20={TOOL_NO 11,BASE_NO 0,IPO_FRAME #BASE,POINT2[] " ",TQ_STATE FALSE}
DECL LDAT LL={VEL 2.00000,ACC 25.0000,APO_DIST 100.000,APO_FAC 50.0000,AXIS_VEL 100.000,AXIS_ACC 100.000,ORI_TYP #VAR,CIRC_TYP #BASE,JERK_FAC 50.0000,GEAR_JERK 50.0000,EXAX_IGN 0}
DECL E6POS XRack_Verde_Pos1={X -982.813232,Y -1660.34290,Z 204.557449,A -90.8999939,B -0.163026243,C -179.937088,S 2,T 42,E1 0.0,E2 0.0,E3 0.0,E4 0.0,E5 0.0,E6 0.0}
DECL FDAT FRack_Verde_Pos1={TOOL_NO 11,BASE_NO 0,IPO_FRAME #BASE,POINT2[] " ",TQ_STATE FALSE}
DECL E6POS XP_aDescarga1_30={X -982.813232,Y -1649.97534,Z 244.090332,A -90.8999939,B -0.163026229,C -179.937088,S 2,T 42,E1 0.0,E2 0.0,E3 0.0,E4 0.0,E5 0.0,E6 0.0}
DECL FDAT FP_aDescarga1_30={TOOL_NO 11,BASE_NO 0,IPO_FRAME #BASE,POINT2[] " ",TQ_STATE FALSE}
DECL E6POS XP_ADESCARGA1_20={X -964.390930,Y -1214.27075,Z 583.063843,A -91.0576630,B -0.170693606,C 179.643661,S 2,T 34,E1 0.0,E2 0.0,E3 0.0,E4 0.0,E5 0.0,E6 0.0}
DECL FDAT FP_aDescarga1_20={TOOL_NO 11,BASE_NO 0,IPO_FRAME #BASE,POINT2[] " ",TQ_STATE FALSE}
DECL E6POS XP_aDescarga1_10={X -964.576416,Y -884.582,Z 977.234,A -90.6960526,B -0.170674115,C 179.643661,S 2,T 34,E1 0.0,E2 0.0,E3 0.0,E4 0.0,E5 0.0,E6 0.0}
DECL FDAT FP_aDescarga1_10={TOOL_NO 11,BASE_NO 0,IPO_FRAME #BASE,POINT2[] " ",TQ_STATE FALSE}
DECL E6POS XRack_Verde_Pos2={X -984.352600,Y -1647.65320,Z 409.716034,A -90.9535294,B -0.0453716330,C -179.888260,S 2,T 42,E1 0.0,E2 0.0,E3 0.0,E4 0.0,E5 0.0,E6 0.0}
DECL FDAT FRack_Verde_Pos2={TOOL_NO 11,BASE_NO 0,IPO_FRAME #BASE,POINT2[] " ",TQ_STATE FALSE}
DECL E6POS XP_aDescarga2_10={X -964.576416,Y -884.582,Z 977.234,A -90.6960526,B -0.170674115,C 179.643661,S 2,T 34,E1 0.0,E2 0.0,E3 0.0,E4 0.0,E5 0.0,E6 0.0}
DECL FDAT FP_aDescarga2_10={TOOL_NO 11,BASE_NO 0,IPO_FRAME #BASE,POINT2[] " ",TQ_STATE FALSE}
DECL E6POS XP_aDescarga2_20={X -964.390930,Y -1214.27075,Z 583.063843,A -91.0576630,B -0.170693606,C 179.643661,S 2,T 34,E1 0.0,E2 0.0,E3 0.0,E4 0.0,E5 0.0,E6 0.0}
DECL FDAT FP_aDescarga2_20={TOOL_NO 11,BASE_NO 0,IPO_FRAME #BASE,POINT2[] " ",TQ_STATE FALSE}
DECL E6POS XP_aDescarga2_30={X -984.352722,Y -1653.19177,Z 442.896179,A -90.9535294,B -0.0453716256,C -179.888260,S 2,T 42,E1 0.0,E2 0.0,E3 0.0,E4 0.0,E5 0.0,E6 0.0}
DECL FDAT FP_aDescarga2_30={TOOL_NO 11,BASE_NO 0,IPO_FRAME #BASE,POINT2[] " ",TQ_STATE FALSE}
DECL E6POS XRack_Verde_Pos3={X -984.924500,Y -1666.06531,Z 617.648254,A -91.1200485,B -0.160327345,C -179.826401,S 2,T 42,E1 0.0,E2 0.0,E3 0.0,E4 0.0,E5 0.0,E6 0.0}
DECL FDAT FRack_Verde_Pos3={TOOL_NO 11,BASE_NO 0,IPO_FRAME #BASE,POINT2[] " ",TQ_STATE FALSE}
DECL E6POS XP_aDescarga3_10={X -964.576416,Y -884.582,Z 977.234,A -90.6960526,B -0.170677662,C 179.643646,S 2,T 34,E1 0.0,E2 0.0,E3 0.0,E4 0.0,E5 0.0,E6 0.0}
DECL FDAT FP_aDescarga3_10={TOOL_NO 11,BASE_NO 0,IPO_FRAME #BASE,POINT2[] " ",TQ_STATE FALSE}
DECL E6POS XP_aDescarga3_20={X -964.459167,Y -1211.52563,Z 816.753906,A -90.6960526,B -0.170677662,C 179.643646,S 2,T 34,E1 0.0,E2 0.0,E3 0.0,E4 0.0,E5 0.0,E6 0.0}
DECL FDAT FP_aDescarga3_20={TOOL_NO 11,BASE_NO 0,IPO_FRAME #BASE,POINT2[] " ",TQ_STATE FALSE}
DECL E6POS XP_aDescarga3_30={X -984.924316,Y -1663.75208,Z 660.453674,A -91.1200485,B -0.160327345,C -179.826401,S 2,T 42,E1 0.0,E2 0.0,E3 0.0,E4 0.0,E5 0.0,E6 0.0}
DECL FDAT FP_aDescarga3_30={TOOL_NO 11,BASE_NO 0,IPO_FRAME #BASE,POINT2[] " ",TQ_STATE FALSE}
DECL E6POS XRack_Verde_Pos4={X -987.065063,Y -1660.26184,Z 831.626099,A -91.0432739,B -0.396091461,C -179.815536,S 2,T 42,E1 0.0,E2 0.0,E3 0.0,E4 0.0,E5 0.0,E6 0.0}
DECL FDAT FRack_Verde_Pos4={TOOL_NO 11,BASE_NO 0,IPO_FRAME #BASE,POINT2[] " ",TQ_STATE FALSE}
DECL E6POS XP_aDescarga4_10={X -970.131653,Y -924.188660,Z 1036.12659,A -90.2109070,B -0.169921443,C 179.636353,S 2,T 34,E1 0.0,E2 0.0,E3 0.0,E4 0.0,E5 0.0,E6 0.0}
DECL FDAT FP_aDescarga4_10={TOOL_NO 11,BASE_NO 0,IPO_FRAME #BASE,POINT2[] " ",TQ_STATE FALSE}
DECL E6POS XP_aDescarga4_20={X -970.063904,Y -1239.25806,Z 879.947571,A -90.2109070,B -0.169924021,C 179.636337,S 2,T 34,E1 0.0,E2 0.0,E3 0.0,E4 0.0,E5 0.0,E6 0.0}
DECL FDAT FP_aDescarga4_20={TOOL_NO 11,BASE_NO 0,IPO_FRAME #BASE,POINT2[] " ",TQ_STATE FALSE}
DECL E6POS XP_aDescarga4_30={X -987.066406,Y -1650.42810,Z 856.247070,A -91.0433350,B -0.396091461,C -179.815536,S 2,T 42,E1 0.0,E2 0.0,E3 0.0,E4 0.0,E5 0.0,E6 0.0}
DECL FDAT FP_aDescarga4_30={TOOL_NO 11,BASE_NO 0,IPO_FRAME #BASE,POINT2[] " ",TQ_STATE FALSE}
DECL E6POS XRack_Verde_Pos5={X -989.027588,Y -1651.36047,Z 1013.22748,A -90.6887741,B -0.445421964,C -179.678314,S 2,T 42,E1 0.0,E2 0.0,E3 0.0,E4 0.0,E5 0.0,E6 0.0}
DECL FDAT FRack_Verde_Pos5={TOOL_NO 11,BASE_NO 0,IPO_FRAME #BASE,POINT2[] " ",TQ_STATE FALSE}
DECL E6POS XP_aDescarga5_10={X -1005.68304,Y -915.485291,Z 1272.16760,A -87.0956650,B -0.164818302,C 179.589554,S 2,T 34,E1 0.0,E2 0.0,E3 0.0,E4 0.0,E5 0.0,E6 0.0}
DECL FDAT FP_aDescarga5_10={TOOL_NO 11,BASE_NO 0,IPO_FRAME #BASE,POINT2[] " ",TQ_STATE FALSE}
DECL E6POS XP_aDescarga5_20={X -973.134216,Y -1230.28516,Z 1099.55652,A -90.7744,B -0.164829254,C 179.589569,S 2,T 34,E1 0.0,E2 0.0,E3 0.0,E4 0.0,E5 0.0,E6 0.0}
DECL FDAT FP_aDescarga5_20={TOOL_NO 11,BASE_NO 0,IPO_FRAME #BASE,POINT2[] " ",TQ_STATE FALSE}
DECL E6POS XP_aDescarga5_30={X -989.027588,Y -1651.36047,Z 1061.75818,A -90.6887741,B -0.445422,C -179.678314,S 2,T 42,E1 0.0,E2 0.0,E3 0.0,E4 0.0,E5 0.0,E6 0.0}
DECL FDAT FP_aDescarga5_30={TOOL_NO 11,BASE_NO 0,IPO_FRAME #BASE,POINT2[] " ",TQ_STATE FALSE}
DECL E6POS XP_SALIDA_RACKVERDE={X -1005.21851,Y -395.575073,Z 1423.46069,A -87.1007538,B -0.167297319,C 179.537186,S 2,T 42,E1 0.0,E2 0.0,E3 0.0,E4 0.0,E5 0.0,E6 0.0}
DECL FDAT FP_SALIDA_RackVerde={TOOL_NO 9,BASE_NO 0,IPO_FRAME #BASE,POINT2[] " ",TQ_STATE FALSE}
DECL PDAT PM={VEL 100.000,ACC 25.0000,APO_DIST 100.000,APO_MODE #CDIS,GEAR_JERK 50.0000,EXAX_IGN 0}
DECL LDAT LM={VEL 2.00000,ACC 25.0000,APO_DIST 100.000,APO_FAC 50.0000,AXIS_VEL 100.000,AXIS_ACC 100.000,ORI_TYP #VAR,CIRC_TYP #BASE,JERK_FAC 50.0000,GEAR_JERK 50.0000,EXAX_IGN 0}
DECL E6POS XP30={X -486.734558,Y -725.266296,Z 1385.97986,A -87.0910187,B -0.133497581,C 179.632736,S 2,T 34,E1 0.0,E2 0.0,E3 0.0,E4 0.0,E5 0.0,E6 0.0}
DECL FDAT FP30={TOOL_NO 11,BASE_NO 0,IPO_FRAME #BASE,POINT2[] " ",TQ_STATE FALSE}
DECL E6POS XP_DROP_1={X -987.400,Y -1664.00,Z 1071.40,A -90.7999878,B -1.00000,C -179.600}
DECL FDAT FP_DROP_1={TOOL_NO 11,BASE_NO 0,IPO_FRAME #BASE,POINT2[] " ",TQ_STATE FALSE}
DECL E6POS XP_DEJAR_AUTO={X 1606.70789,Y -354.796814,Z 1944.22656,A 1.33749425,B -32.3921471,C 179.037674,S 2,T 42,E1 0.0,E2 0.0,E3 0.0,E4 0.0,E5 0.0,E6 0.0}
DECL FDAT FP_DEJAR_AUTO={TOOL_NO 11,BASE_NO 0,IPO_FRAME #BASE,POINT2[] " ",TQ_STATE FALSE}
DECL E6POS XP_DEJAR_VERDE={X -987.400,Y -1664.00,Z 991.400,A -90.7999878,B -1.00000,C -179.600}
DECL FDAT FP_DEJAR_VERDE={TOOL_NO 11,BASE_NO 0,IPO_FRAME #BASE,POINT2[] " ",TQ_STATE FALSE}
DECL E6POS XP_DROP_2={X -987.400,Y -1664.00,Z 1071.40,A -90.7999878,B -1.00000,C -179.600}
DECL FDAT FP_DROP_2={TOOL_NO 11,BASE_NO 0,IPO_FRAME #BASE,POINT2[] " ",TQ_STATE FALSE}
DECL E6POS XP_DROP_3={X -987.400,Y -1664.00,Z 1071.40,A -90.7999878,B -1.00000,C -179.600}
DECL FDAT FP_DROP_3={TOOL_NO 11,BASE_NO 0,IPO_FRAME #BASE,POINT2[] " ",TQ_STATE FALSE}
DECL E6POS XP_DROP_4={X -987.400,Y -1664.00,Z 1071.40,A -90.7999878,B -1.00000,C -179.600}
DECL FDAT FP_DROP_4={TOOL_NO 11,BASE_NO 0,IPO_FRAME #BASE,POINT2[] " ",TQ_STATE FALSE}
DECL E6POS XP_DROP_5={X -987.400,Y -1664.00,Z 1071.40,A -90.7999878,B -1.00000,C -179.600}
DECL FDAT FP_DROP_5={TOOL_NO 11,BASE_NO 0,IPO_FRAME #BASE,POINT2[] " ",TQ_STATE FALSE}
DECL E6POS XP_Espera_Dejar_Rack_V={X -1005.80304,Y -559.825378,Z 1414.28723,A -87.0956573,B -0.164799362,C 179.589539,S 2,T 34,E1 0.0,E2 0.0,E3 0.0,E4 0.0,E5 0.0,E6 0.0}
DECL FDAT FP_Espera_Dejar_Rack_V={TOOL_NO 11,BASE_NO 0,IPO_FRAME #BASE,POINT2[] " ",TQ_STATE FALSE}
DECL E6POS XPOS_ESPERA_RACK_VERDE={X 772.101379,Y -764.727417,Z 1373.18774,A -87.1007538,B -0.167297110,C 179.537186,S 2,T 34,E1 0.0,E2 0.0,E3 0.0,E4 0.0,E5 0.0,E6 0.0}
DECL FDAT FPOS_ESPERA_RACK_VERDE={TOOL_NO 11,BASE_NO 0,IPO_FRAME #BASE,POINT2[] " ",TQ_STATE FALSE}
DECL PDAT PL={VEL 100.000,ACC 25.0000,APO_DIST 100.000,GEAR_JERK 50.0000,EXAX_IGN 0}
ENDDAT
